FUNCTION_BLOCK FB_Scaling
VAR_INPUT
	nRawInputValue			: INT;
	nInputLowerLimit		: INT;
	nInputHigherLimit		: DINT;
	nOutputLowerLimit		: LREAL;
	nOutputHigherLimit		: LREAL;
END_VAR
VAR_OUTPUT 
		nScaledValueF		: LREAL;
	    nScaledValueD		: INT;
END_VAR
VAR
	 nGain		: REAL;
	Temp: STRING(510);
END_VAR

// Scaling Calculations //

	IF	nRawInputValue	<	0	THEN
		nRawInputValue	:=	0;
	END_IF


	IF	 ((nInputHigherLimit - nInputLowerLimit)	<= 0)	THEN
//		 ((nOutputHigherLimit  - nOutputLowerLimit)	<= 0)	THEN
		nGain	:=	0;
	ELSE
//				nGain:=(((nRawInputValue - nInputLowerLimit) / (nInputHigherLimit - nInputLowerLimit)) * (nOutputHigherLimit  - nOutputLowerLimit)) + nOutputLowerLimit;
		nGain:=(nRawInputValue - nInputLowerLimit)*((nOutputHigherLimit - nOutputLowerLimit) / (nInputHigherLimit - nInputLowerLimit)) + nOutputLowerLimit;
	END_IF


		Temp	:=	LREAL_TO_FMTSTR( nGain, 1, TRUE );
		
		nScaledValueF	:=	STRING_TO_REAL(Temp);
		nScaledValueD	:=	REAL_TO_INT(nGain);

END_FUNCTION_BLOCK

(* stored: Version 1.1.0.1, ProductVersion 3.1.4024.9
   POU FB_Scaling: Id {9d98f2c2-045a-45d7-a8db-68b4e460594c}, SpecialFunc None *)
